{attribute 'GeneratedUsingTerminal: ELX3252-0000-0016'}
{attribute addProperty BoxType "ELX3252-0000-0016"}
{attribute addProperty Id "Limit_1BYTE1Limit_2BYTE1ErrorBOOL1TxPDO_StateBOOL1TxPDO_ToggleBOOL1"}
{attribute addProperty CRC "2924311467"}
{attribute addProperty Size "5"}
TYPE Status_AE4D73AB :
STRUCT
	{attribute addProperty Name "Limit_1"}
	Limit_1 : BYTE;
	{attribute addProperty Name "Limit_2"}
	Limit_2 : BYTE;
	{attribute addProperty Name "Error"}
	Error : BOOL;
	{attribute addProperty Name "TxPDO_State"}
	TxPDO_State : BOOL;
	{attribute addProperty Name "TxPDO_Toggle"}
	TxPDO_Toggle : BOOL;
END_STRUCT
END_TYPE

(* stored: Version 1.2.0.0, ProductVersion 3.1.4024.9
   DUT Status_AE4D73AB: Id {638ffdc0-7217-40e8-89d8-bc4937841bd5} *)
